{attribute 'obsolete' := 'Use FB_PositionState1D_InOut instead'}
FUNCTION_BLOCK FB_PositionStateInOut EXTENDS FB_PositionStateBase
(*
    Example usage of FB_PositionStateBase for a simple IN/OUT axis. See NOTE: comments.
    Also usable as a drop-in for these cases (no need to roll your own in/out)
*)
VAR_INPUT
    // The enum position to move to
    {attribute 'pytmc' := '
        pv: SET
        io: io
    '}
    enumSet: ENUM_EpicsInOut_INT; // NOTE: Please copy this pragma exactly on your enumSet

    // Information about the OUT position
    stOut: ST_PositionState; // NOTE: Do not pragma these, let it happen in the manager.
    // Information about the IN position
    stIn: ST_PositionState;
END_VAR
VAR_OUTPUT
    // The enum state readback
    {attribute 'pytmc' := '
        pv: GET
        io: i
    '}
    enumGet: ENUM_EpicsInOut_INT; // NOTE: Please copy this pragma exactly on your enumGet
END_VAR
VAR
    bInOutInit: BOOL;
END_VAR


IF NOT bInOutInit THEN
    bInOutInit := TRUE;
    arrStates[1] := stOut;
    arrStates[2] := stIn;
    stOut.sName := 'OUT';
    stIn.sName := 'IN';
END_IF
setState := enumSet;
Exec();
enumGet := getState;
enumSet := setState;

END_FUNCTION_BLOCK

(* stored: Version 1.1.0.1
   POU FB_PositionStateInOut: Id {0410dcaa-d262-4dff-9ed9-0476e0f72083}, SpecialFunc None *)
